FUNCTION_BLOCK FB_Enabled
VAR_INPUT
END_VAR
VAR_OUTPUT
END_VAR
VAR
END_VAR

	IF HMIinput.bHMIOnOffSwitch = FALSE THEN // When on-off switch is OFF
		
		HMIoutput.bHMIRedLED := FALSE;	// Red light cant be on
	
	ELSIF HMIinput.bHMIOnOffSwitch = TRUE AND HMIinput.bHMIStartSwitch = FALSE THEN // When on-off is on and the start switch is off
	
		HMIoutput.bHMIRedLED := TRUE;	// Red light is on
		
	END_IF
	
	
	
	
	IF HMIinput.bHMIStopSwitch = TRUE THEN 	// When stop switch is on
		
		HMIinput.bHMIStartSwitch := FALSE;	// Start switch is off
		
		HMIinput.bHMIStopSwitch := FALSE;	// Stop switch is off
	
	END_IF
	
	
	
	IF HMIinput.bHMIStartSwitch = TRUE THEN	// When start switch is on
		
		HMIoutput.bHMIGreenLED := TRUE;		// Green light is on
		
		HMIoutput.bHMIRedLED := FALSE;		// Red light is off
	
	ELSE									// When start switch is off
		
		HMIoutput.bHMIGreenLED := FALSE;	// Green light is off
	
	END_IF

END_FUNCTION_BLOCK

(* stored: Version 1.1.0.1, ProductVersion 3.1.4024.10
   POU FB_Enabled: Id {62224dc0-3d97-4153-b94c-f43bb0472034}, SpecialFunc None *)
